    # Documented in monorepo/doc/pal/PalAdvancedProgrammingFunctions.md
    def rq_set_conveyor_clearance(is_left_pallet, height):
      if height < 0:
        popup("rq_set_conveyor_clearance(): The clearance height should be positive.", title="Palletizer", error=True,
        blocking=True)
      elif height == 0:
        height = 0.0001
      end

      pallet_side = "right"
      if(is_left_pallet):
         pallet_side = "left"
      end

      local palletId = node_rpc_server.getPalletId(pallet_side)
      node_rpc_server.setConveyorVerticalClearance(palletId, height)
    end
    ###############################################################
    # Linear Axis Move related methods
    ###############################################################
    def verify_is_in_linear_axis_range(target_axis_position):
      axis_position_range = node_rpc_server.linearaxisgetpositionrange()

      if target_axis_position < axis_position_range[0] or target_axis_position > axis_position_range[1]:
        textmsg("Linear axis target position : ", target_axis_position)
        textmsg("Linear axis position range : ", axis_position_range)
        popup("Linear axis position is unreachable.", "Linear Axis Move", blocking=True, error=True)
        halt
      end
    end

    # Documented in monorepo/doc/pal/PalAdvancedProgrammingFunctions.md
    def rq_get_linear_axis_pos():
        axis_position = node_rpc_server.linearaxisgetactualposition()
        return axis_position
    end

  BLOW_OFF_MODE_NO_AIR = 0
  BLOW_OFF_MODE_SMART_AIR = 1
  UNDEFINED_THREAD_ID = -1
  MODBUS_TYPE = "MODBUS"
  STANDARD_TYPE = "STANDARD"
  INVALID_OUTPUT_ADDRESS = -1
  RQ_UNUSED_TIMEOUT = -1

  global rq_cnc_insertion_node_ids = [-1, -1]
  global rq_run_timeout = 30

  ###################################################################################
  #
  # Generic methods
  #
  ###################################################################################

  def bool_to_str(value):
    if value:
      return "true"
    else:
      return "false"
    end
  end

  def bool_array_to_string(array, index):
    if (index >= length(array)):
      return "]"
    end

    separator = ","
    if (index == length(array) - 1):
      separator = ""
    end

    if (index == 0):
      str_array = concat("[", bool_to_str(array[index]), separator)
      return str_cat(str_array, bool_array_to_string(array, index + 1))
    else:
      return concat(bool_to_str(array[index]), separator, bool_array_to_string(array, index + 1))
    end
  end

  def rq_bool_array_to_string(array):
    return bool_array_to_string(array, 0)
  end

  def json_force_node(force, max_negative_deviation, max_positive_deviation, stiffness, enabled_axis, feature, is_adaptive):
    json = "{"
    json = concat(json, key_val("forceFrame", feature), ",")
    json = concat(json, key_val("isAdaptive", is_adaptive), ",")
    json = concat(json, key_val("isForceControlAboutActualPosition", "false"), ",")
    json = concat(json, key_val("isForceMode", enabled_axis), ",")
    json = concat(json, key_val("maxNegativeDeviation", max_negative_deviation), ",")
    json = concat(json, key_val("maxPositiveDeviation", max_positive_deviation), ",")
    json = concat(json, key_val("stiffness", stiffness), ",")
    json = concat(json, key_val("targetTcpWrench", force), "}")
    return json
  end

  def rq_setup_machine_tending_force_node(feature, force, stiffness, max_negative_deviation, max_positive_deviation, enabled_axis, is_adaptive):
    force_node_id = node_rpc_server.createnewforcenode()
    node_rpc_server.fromjson(force_node_id, json_force_node(force, max_negative_deviation, max_positive_deviation,
    stiffness, rq_bool_array_to_string(enabled_axis), 1, bool_to_str(is_adaptive)))
    return force_node_id
  end

  ###################################################################################
  #
  # TRAJECTORY UTILITIES
  #
  ###################################################################################

  def dot_product(v1, v2):
    return [v1]*transpose(v2)
  end

  def get_symmetric_poses_from_middle(p1, p2, middle_pose, distance):
    distance_p1_middle = point_dist(p1, middle_pose)
    alpha = (distance / 2) / distance_p1_middle
    start_pose = interpolate_pose(middle_pose, p1, alpha)
    end_pose = interpolate_pose(middle_pose, p2, alpha)

    return [start_pose, end_pose]
  end

  def translate_to_origin(pose):
    return p[0, 0, 0, pose[3], pose[4], pose[5]]
  end


  ###################################################################################
  #
  # ROBOTIQ PART PRESENTER
  #
  ###################################################################################

  global cnc_part_presenter_index = 0

  def rq_pallet_get_poses_from_index(p_corner_1_approach, p_corners, nb_rows, nb_columns, alternate_direction, index):
      row = floor(index / nb_columns)
      column = index % nb_columns

      row_alpha = 0
      if(nb_rows > 1):
          row_alpha = row / (nb_rows - 1)
      end

      p_row_start = interpolate_pose(p_corners[0], p_corners[3], row_alpha)
      p_row_end = interpolate_pose(p_corners[1], p_corners[2], row_alpha)

      column_alpha = 0
      if(nb_columns > 1):
          column_alpha = column / (nb_columns - 1)
      end

      if(alternate_direction and (row % 2) and nb_columns > 1):
          pallet_pose = interpolate_pose(p_row_end, p_row_start, column_alpha)
      else:
          pallet_pose = interpolate_pose(p_row_start, p_row_end, column_alpha)
      end

      T_1approach_1 = pose_trans(inv(p_corner_1_approach), p_corners[0])
      approach_pose = pose_trans(pallet_pose, inv(T_1approach_1))

      return [approach_pose, pallet_pose]
  end

  ###################################################################################
  #
  # MOVE DOOR
  #
  ###################################################################################

  def rq_setup_door_force_node(reference_frame, force, stiffness):
    feature = 1
    forces = [force,0,0,0,0,0]
    max_negative_deviation = [-5, 0, 0, 0, 0, 0]
    max_positive_deviation = [0.01, 0, 0, 0, 0, 0] # using a large value here would allow the trajectory to violate the kinematics limits, using zero removes the force node effect
    stiffnesses = [stiffness, 100, 100, 100, 100, 100]
    enabled_axis = [True, False, False, False, False, False]
    is_adaptive = True

    force_node_id = rq_setup_machine_tending_force_node(feature, forces, stiffnesses, max_negative_deviation,
    max_positive_deviation, enabled_axis, is_adaptive)

    node_rpc_server.setCustomFixedForceFrame(force_node_id, [reference_frame[3],reference_frame[4],reference_frame[5]])

    return force_node_id
  end

  def json_rq_moves_node(tcp_speed, tcp_accel):
    json = "{"
    json = concat(json, key_val("offsetType", 0), ",")
    json = concat(json, key_val("tcpSpeed", tcp_speed), ",")
    json = concat(json, key_val("tcpAccel", tcp_accel), ",")
    json = concat(json, key_val("actualreferenceframe", [0, 0, 0, 0, 0, 0]), ",")
    json = concat(json, key_val("originalreferenceframe", [0, 0, 0, 0, 0, 0]), "}")
    return json
  end

  def rq_setup_rqmoves_node(parent_node_id, tcp_speed, tcp_accel):
    rq_moves_node_id = node_rpc_server.createnewrqmoves()
    node_rpc_server.fromjson(rq_moves_node_id, json_rq_moves_node(tcp_speed, tcp_accel))
    node_rpc_server.setparentid(rq_moves_node_id, parent_node_id)
    return rq_moves_node_id
  end

  def rq_setup_waypoint_node(pose, joints, is_straight, parent_node_id):
    def json_waypoint_node(pose, joints, is_straight):
      json = "{"
      json = concat(json, key_val("jointPositions", joints), ",")
      json = concat(json, key_val("tcpPose", [pose[0],pose[1],pose[2],pose[3],pose[4],pose[5]]), ",")
      json = concat(json, key_val("isStraight", bool_to_str(is_straight)), "}")
      return json
    end

    waypoint_node_id = node_rpc_server.createnewwaypointnode()
    node_rpc_server.fromjson(waypoint_node_id, json_waypoint_node(pose, joints, is_straight))
    node_rpc_server.setparentid(waypoint_node_id, parent_node_id)
    node_rpc_server.rqmovesaddwaypoint(parent_node_id, waypoint_node_id)
    return waypoint_node_id
  end

  def rq_setup_move_door(reference_frame, start_pose, start_joints, stop_pose, stop_joints, move_force, contact_force, tcp_speed=0.4, tcp_accel=0.4):

    stop_pose_in_start_frame = pose_trans(pose_inv(start_pose), stop_pose)

    seeks_contact = False
    stiffness = 10
    move_force_node_id = rq_setup_door_force_node(reference_frame, move_force, stiffness)
    rq_moves_node_id = rq_setup_rqmoves_node(move_force_node_id, tcp_speed, tcp_accel)
    waypoint_open = rq_setup_waypoint_node(start_pose, start_joints, False, rq_moves_node_id)
    waypoint_close = rq_setup_waypoint_node(stop_pose, stop_joints, True, rq_moves_node_id)
    seeks_contact = True
    stiffness = 100
    contact_force_node_id = rq_setup_door_force_node(reference_frame, contact_force, stiffness)

    rq_movej_node_id = node_rpc_server.createnewmovejnode()
    node_rpc_server.setparentid(rq_movej_node_id, move_force_node_id)

    return [move_force_node_id, rq_moves_node_id, waypoint_open, waypoint_close, contact_force_node_id, rq_movej_node_id]
  end

  def rq_move_door(start_pose, start_joints, stop_pose, stop_joints, move_force, contact_force, tcp_speed, tcp_accel, approach_pose, approach_joints, end_reached_threshold=0.001):

    reference_frame = list_to_pose(kinematics_rpc_server.reorientP1WithXTowardP2andZApproxP1Z(start_pose, stop_pose))

    node_ids = rq_setup_move_door(reference_frame, start_pose, start_joints, stop_pose, stop_joints, move_force, contact_force, tcp_speed, tcp_accel)

    move_force_node_id = node_ids[0]
    rq_moves_node_id = node_ids[1]
    start_waypoint_node_id = node_ids[2]
    end_waypoint_node_id = node_ids[3]
    contact_force_node_id = node_ids[4]
    rq_movej_node_id = node_ids[5]

    rq_wait_ft_sensor_steady(2000)
    zero_ftsensor()
    sleep(0.1)

    path_answer = node_rpc_server.rqmovesinit(rq_moves_node_id)
    verify_path_answer(path_answer)

    approach_position_joints = get_inverse_kin(approach_pose, qnear=approach_joints)
    movej(approach_position_joints)

    node_rpc_server.movejdefinewaypoint(rq_movej_node_id, get_actual_joint_positions(), 1.0, 1.0)
    node_rpc_server.setparentid(rq_movej_node_id, move_force_node_id)
    reset_node_executor()
    active_and_reset_node(move_force_node_id)
    node_execution_thread = execute_node(rq_movej_node_id, True)

    path_answer = node_rpc_server.rqmovesinit(rq_moves_node_id)
    verify_path_answer(path_answer)
    q0 = node_rpc_server.rqmovesgetfirstpoint(rq_moves_node_id)
    node_rpc_server.setparentid(rq_movej_node_id, move_force_node_id)
    node_rpc_server.movejdefinewaypoint(rq_movej_node_id, q0, 1.0, 0.4)
    execute_node(rq_movej_node_id)
    execute_node(start_waypoint_node_id)
    execute_node(end_waypoint_node_id)

    kill_thread(node_execution_thread)

    node_rpc_server.movejdefinewaypoint(rq_movej_node_id, get_actual_joint_positions(), 1.0, 1.0)
    node_rpc_server.setparentid(rq_movej_node_id, contact_force_node_id)
    reset_node_executor()
    active_and_reset_node(contact_force_node_id)
    node_execution_thread = execute_node(rq_movej_node_id, True)

    timeout = 20
    while (point_dist(get_actual_tcp_pose(), stop_pose) > end_reached_threshold):
      if (timeout <= 0):
        popup("Door has not reached its final position")
        halt
      else:
        sync()
        timeout = timeout - get_steptime()
      end
    end

    kill_thread(node_execution_thread)

    approach_pose_in_start_frame = pose_trans(pose_inv(start_pose), approach_pose)
    retract_pose = pose_trans(get_actual_tcp_pose(), approach_pose_in_start_frame)
    movej(retract_pose)

    node_rpc_server.deletenode(move_force_node_id)
    node_rpc_server.deletenode(rq_moves_node_id)
    node_rpc_server.deletenode(start_waypoint_node_id)
    node_rpc_server.deletenode(end_waypoint_node_id)
    node_rpc_server.deletenode(contact_force_node_id)
    node_rpc_server.deletenode(rq_movej_node_id)

  end

  ###################################################################################
  #
  # CNC Insertion
  #
  ###################################################################################

  def rq_collet_insertion(contact_pose, insert_pose, inserted_pose):
      movel(contact_pose, a=1.2, v=0.025)
      movel(insert_pose, a=1.2, v=0.025)

      zero_ftsensor()
      sleep(0.1)

      direction = "Z+"
      stop_force_threshold = 3.0
      max_radius = 5.0
      radius_incr = 0.7
      peck_mode = False
      tangential_speed = 0.02
      compliant_insert_force_threshold = 10.0
      spiral_initial_pose_offset_name = "spiral_initial_pose_offset_name"
      rq_ins_destination = inserted_pose
      max_distance = point_dist(inserted_pose, get_actual_tcp_pose())
      rq_spiral_not_completed = False
      rq_ins_speed_setting = 0.02

      rq_insert_spiral_urcap(direction, stop_force_threshold, max_radius, radius_incr, peck_mode, tangential_speed, compliant_insert_force_threshold, spiral_initial_pose_offset_name)

      if (rq_spiral_not_completed):
        return False
      end

      return True
  end

  def rq_push_part(approach_pose, chuck_pose):
      zero_ftsensor()
      sleep(0.1)

      # Find pose with z axis pointing in the direction of the insertion
      p1 = translate_to_origin(approach_pose)
      insertion_dir_in_base_frame = pose_trans(p1, pose_trans(pose_inv(approach_pose), chuck_pose))
      ref_frame_pose = list_to_pose(kinematics_rpc_server.poseFromZaxis([insertion_dir_in_base_frame[0], insertion_dir_in_base_frame[1], insertion_dir_in_base_frame[2]]))

      surface_found = rq_linear_search_custom_frame("Z+", 10.0, 0.025, 0.1, ref_frame_pose)

      if not(surface_found):
          return False
      end

      return True
  end

  def rq_place_in_chuck(close_chuck_do, open_chuck_do, chuck_approach, chuck_position, chuck_delay):
      rq_open_workholding(close_chuck_do, open_chuck_do)

      movel(chuck_approach, a=1.2, v=0.25)
      movel(chuck_position, a=1.2, v=0.25)

      rq_close_workholding(close_chuck_do, open_chuck_do)
      sleep(chuck_delay)
  end

  def rq_pre_pick_in_chuck(chuck_approach, chuck_position, speed=0.25, accel=1.2):
      movel(chuck_approach, accel, speed)
      movel(chuck_position, accel, speed)
  end

  def rq_post_pick_in_chuck(close_chuck_do, open_chuck_do, chuck_approach, chuck_position, chuck_delay, speed=0.25,
  accel=1.2):
      rq_open_workholding(close_chuck_do, open_chuck_do)
      sleep(chuck_delay)

      movel(chuck_approach, accel, speed)
  end

  def rq_open_workholding(close_do, open_do):
      rq_set_workholding_do(close_do, open_do, False)
  end

  def rq_close_workholding(close_do, open_do):
      rq_set_workholding_do(close_do, open_do, True)
  end

  def rq_set_workholding_do(close_do, open_do, close_request):
      is_close_do_valid = rq_is_do_valid(close_do)
      is_open_do_valid = rq_is_do_valid(open_do)

      if(is_close_do_valid):
          set_standard_digital_out(close_do, close_request)
      end
      if(is_open_do_valid):
          set_standard_digital_out(open_do, not close_request)
      end
      if(is_close_do_valid or is_open_do_valid):
          sleep(0.5)
      end
  end

  def rq_is_do_valid(do_id):
      return do_id >= 0 and do_id <= 7
  end

  def set_cleaning_digital_output(address, state, blow_off_mode, output_type):
     if(blow_off_mode == BLOW_OFF_MODE_SMART_AIR):
       rq_set_output(output_type, address, state)
     end
  end

  ###################################################################################
  #
  # PATH GENERATOR 6 POINTS CURVE BUILT WITH 2 POINTS
  #
  ###################################################################################

  def execute_half_pipe(pose_1, pose_2,pose_transformation_air_nozzle_to_actual_tcp, depth, length_distance, width, angle, speed, spacing, address, output_type, blow_off_mode, passes):
    path_gen_poses = get_path_generator_6_points_poses(pose_1, pose_2, pose_transformation_air_nozzle_to_actual_tcp, depth, length_distance, width, angle)
    start_pose = p[path_gen_poses[0,0],path_gen_poses[0,1],path_gen_poses[0,2],path_gen_poses[0,3],path_gen_poses[0,4],path_gen_poses[0,5]]
    path_generator_node_id = setup_path_generator_6_points(path_gen_poses, speed, spacing)
    execute_path_generator_6_points(path_generator_node_id, start_pose,  address, output_type, blow_off_mode, passes)
  end

  def get_path_generator_6_points_poses(pose_2, pose_5,pose_transformation_air_nozzle_to_actual_tcp, depth=0.01, length=0, width=0.05, angle_deg=0):

    def offset_pose(pose, offset, offset_reference_frame, pose_transformation_air_nozzle_to_actual_tcp):
      pose_relative_to_ref_frame = express_pose_A_relative_to_pose_B(pose, offset_reference_frame)
      ref_frame_with_offset = pose_trans(offset_reference_frame, offset)
      pose_with_offset = pose_trans(ref_frame_with_offset, pose_relative_to_ref_frame)
      pose_with_offset_for_actual_tcp = pose_trans(pose_with_offset, pose_transformation_air_nozzle_to_actual_tcp)
      return pose_to_list(pose_with_offset_for_actual_tcp)
    end

    if(length > 0):
      middle_pose = interpolate_pose(pose_2, pose_5, 0.5)

      poses = get_symmetric_poses_from_middle(pose_2, pose_5, middle_pose, length)
      pose_2 = poses[0]
      pose_5 = poses[1]
    end

    path_ref_frame = list_to_pose(kinematics_rpc_server.reorientP1WithXTowardP2andZApproxP1Z(pose_2, pose_5))

    offset1 = pose_add(p[0,0,0,0,d2r(angle_deg),0], p[0, width,-depth,-d2r(angle_deg),0,0])
    offset2 = pose_add(p[0,0,0,0,d2r(angle_deg),0], p[0,     0,     0,              0,0,0])
    offset3 = pose_add(p[0,0,0,0,d2r(angle_deg),0], p[0,-width,-depth, d2r(angle_deg),0,0])

    pose_1_array = offset_pose(pose_2, offset1, path_ref_frame, pose_transformation_air_nozzle_to_actual_tcp)
    pose_2_array = offset_pose(pose_2, offset2, path_ref_frame, pose_transformation_air_nozzle_to_actual_tcp)
    pose_3_array = offset_pose(pose_2, offset3, path_ref_frame, pose_transformation_air_nozzle_to_actual_tcp)

    pose_4_array = offset_pose(pose_5, offset1, path_ref_frame, pose_transformation_air_nozzle_to_actual_tcp)
    pose_5_array = offset_pose(pose_5, offset2, path_ref_frame, pose_transformation_air_nozzle_to_actual_tcp)
    pose_6_array = offset_pose(pose_5, offset3, path_ref_frame, pose_transformation_air_nozzle_to_actual_tcp)

    return [pose_1_array, pose_2_array, pose_3_array, pose_4_array, pose_5_array, pose_6_array]
  end

  def setup_path_generator_6_points(pose_list, tcp_speed=0.1, spacing=0.02):

    def json_path_generator_node(pose_list, tcp_speed, spacing):

      SIX_POINTS_CURVE = 3
      OFFSET_TYPE_NONE = 0
      FORCE_OPPOSITE_SIDE = 2

      json = "{"
      json = concat(json, key_val("tcpSpeed", tcp_speed), ",")
      json = concat(json, key_val("poses", pose_list), ",")
      json = concat(json, key_val("avoidAbruptEnd", "false"), ",")
      json = concat(json, key_val("isSurfaceFillOn", "true"), ",")
      json = concat(json, key_val("spacing", spacing), ",")
      json = concat(json, key_val("pathType", SIX_POINTS_CURVE), ",")
      json = concat(json, key_val("offsetType",OFFSET_TYPE_NONE), ",")
      json = concat(json, key_val("endingMode", FORCE_OPPOSITE_SIDE), "}")

      return json
    end

    rq_path_generator_parent_id = 0
    path_generator_node_id = node_rpc_server.createPathGeneratorNode()
    node_rpc_server.fromjson(path_generator_node_id, json_path_generator_node(pose_list, tcp_speed, spacing))
    node_rpc_server.setparentid(path_generator_node_id, rq_path_generator_parent_id)

    return path_generator_node_id
  end

  def execute_path_generator_6_points(path_generator_node_id, pose_1, address = INVALID_OUTPUT_ADDRESS, output_type = MODBUS_TYPE, blow_off_mode = BLOW_OFF_MODE_NO_AIR, passes = 1):
    index = 0
    while (index < passes):
      movej(get_inverse_kin(pose_1))
      set_cleaning_digital_output(address, True, blow_off_mode, output_type)
      reset_node_executor()
      node_execution_thread = execute_node(path_generator_node_id, True)
      rq_continue_node_execution = False
      set_cleaning_digital_output(address, False, blow_off_mode, output_type)
      join node_execution_thread
      index = index + 1
    end
    node_rpc_server.deletenode(path_generator_node_id)
  end

  ###################################################################################
  #
  # Straight line trajectory
  #
  ###################################################################################

  def execute_straight_line(p1, p2,pose_transformation_air_nozzle_to_actual_tcp, accel=1.2, speed=0.25, distance = 0, angles = [0, 0, 0], address = INVALID_OUTPUT_ADDRESS, output_type = MODBUS_TYPE, blow_off_mode = BLOW_OFF_MODE_NO_AIR, passes = 1):
    offset_for_angles = p[0, 0, 0, d2r(angles[0]), d2r(angles[1]), d2r(angles[2])]
    p1 = pose_trans(p1, offset_for_angles)
    p2 = pose_trans(p2, offset_for_angles)

    # apply transformation to take into account that the actual tcp offset is not the same as the one that was used when the waypoints were saved:
    p1 = pose_trans(p1, pose_transformation_air_nozzle_to_actual_tcp)
    p2 = pose_trans(p2, pose_transformation_air_nozzle_to_actual_tcp)
    global air_output_adress = address

    qActual = get_actual_joint_positions()
    CleanPathId = node_rpc_server.createnewcleaningpathnode(p1, p2, qActual, passes, distance, accel, speed, blow_off_mode)

    reset_node_executor()
    if output_type == MODBUS_TYPE:
      air_thread = run modbusAirControlThread()
    elif output_type == STANDARD_TYPE:
      air_thread = run standardAirControlThread()
    end

    node_execution_thread = execute_node(CleanPathId, True)
    rq_continue_node_execution = False

    join node_execution_thread
    node_rpc_server.deletenode(CleanPathId)
    if output_type == MODBUS_TYPE or output_type == STANDARD_TYPE :
      kill air_thread
    end
  end

  ###################################################################################
  #
  # Cross trajectory
  #
  ###################################################################################

  def find_cross_trajectory_poses(p1, p2, height=0, width=0, p1_angles = [0, 0, 0], p2_angles = [0, 0, 0], p3_angles = [0, 0, 0], p4_angles = [0, 0, 0]):
    def find_side_poses(p0, p1):
      def find_side_pose(p0,p1,angle):
        p1_T_p0 = pose_trans(pose_inv(p0), p1)
        rotated_p0_by_90_degrees = pose_trans(p0, p[0, 0, 0, 0, 0, d2r(angle)])

        side_pose = pose_trans(rotated_p0_by_90_degrees, p1_T_p0)
        side_pose[3] = p0[3]
        side_pose[4] = p0[4]
        side_pose[5] = p0[5]

        return side_pose
      end

      p3= find_side_pose(p0, p1, 90)
      p4 = find_side_pose(p0, p1, 270)

      return [p3, p4]
    end

    def get_start_and_end_poses_based_on_distance(p1, p2, middle_pose, distance):
      if(distance == 0):
        start_pose = p1
        end_pose = p2
      else:
        poses = get_symmetric_poses_from_middle(p1, p2, middle_pose, distance)
        start_pose = poses[0]
        end_pose = poses[1]
      end
      return [start_pose, end_pose]
    end

    def get_side_poses_based_on_distance(p1, p2, middle_pose, width):
      if(width == 0):
        side_poses = find_side_poses(middle_pose, p1)
      else:
        poses = get_symmetric_poses_from_middle(p1, p2, middle_pose, width)
        side_poses = find_side_poses(middle_pose, poses[0])
      end

      return side_poses
    end

    def get_angle_offset(angles):
      return  p[0, 0, 0, d2r(angles[0]), d2r(angles[1]), d2r(angles[2])]
    end

    middle_pose = interpolate_pose(p1, p2, 0.5)

    start_and_end_poses = get_start_and_end_poses_based_on_distance(p1, p2, middle_pose, height)
    side_poses = get_side_poses_based_on_distance(p1, p2, middle_pose, width)

    p1_offset = get_angle_offset(p1_angles)
    p2_offset = get_angle_offset(p2_angles)
    p3_offset = get_angle_offset(p3_angles)
    p4_offset = get_angle_offset(p4_angles)

    start_and_end_poses[0] = pose_trans(start_and_end_poses[0], p1_offset)
    start_and_end_poses[1] = pose_trans(start_and_end_poses[1], p2_offset)
    side_poses[0] = pose_trans(side_poses[0], p3_offset)
    side_poses[1] = pose_trans(side_poses[1], p4_offset)

    return [middle_pose, start_and_end_poses[0], start_and_end_poses[1], side_poses[0], side_poses[1]]
  end

  def execute_cross_trajectory(p1, p2,pose_transformation_air_nozzle_to_actual_tcp, height=0, width=0, p1_angles = [0, 0, 0], p2_angles = [0, 0, 0], p3_angles = [0, 0, 0], p4_angles = [0, 0, 0], accel=1.2, speed=0.25,  address = INVALID_OUTPUT_ADDRESS, output_type = MODBUS_TYPE, blow_off_mode = BLOW_OFF_MODE_NO_AIR, passes = 1):

    cross_poses = find_cross_trajectory_poses(p1, p2, height, width, p1_angles, p2_angles, p3_angles, p4_angles)

    p0 = pose_trans(cross_poses[0], pose_transformation_air_nozzle_to_actual_tcp)
    p1 = pose_trans(cross_poses[1], pose_transformation_air_nozzle_to_actual_tcp)
    p2 = pose_trans(cross_poses[2], pose_transformation_air_nozzle_to_actual_tcp)
    p3 = pose_trans(cross_poses[3], pose_transformation_air_nozzle_to_actual_tcp)
    p4 = pose_trans(cross_poses[4], pose_transformation_air_nozzle_to_actual_tcp)

   index = 0

   while (index < passes):
     movej(get_inverse_kin(p0))
     set_cleaning_digital_output(address, True, blow_off_mode, output_type)
     movel(p1, accel, speed)
     movel(p2, accel, speed)
     movel(p0, accel, speed)
     movel(p3, accel, speed)
     movel(p4, accel, speed)
     set_cleaning_digital_output(address, False, blow_off_mode, output_type)
     index = index + 1
   end
  end

  def execute_waypoint_cross_trajectory(starting_pose, finishing_pose, accel=1.2, speed=0.25):
   movej(get_inverse_kin(starting_pose))
   movel(finishing_pose, accel, speed)
  end

  ###################################################################################
  #
  # Fermat spiral trajectory
  #
  ###################################################################################

  def execute_fermat_spiral(start_pose, end_pose,pose_transformation_air_nozzle_to_actual_tcp, max_radius = 0, angle = 0, number_of_turns = 1, speed = 0.25,address = INVALID_OUTPUT_ADDRESS, output_type = MODBUS_TYPE, blow_off_mode = BLOW_OFF_MODE_NO_AIR, passes = 1):
    def find_middle(start_pose, end_pose):
      alpha = 0.5
      return interpolate_pose(start_pose, end_pose, alpha)
    end

    def find_next_theta(spiral_constant, theta, speed):
      denom = spiral_constant * sqrt(1/(4*theta) + theta)
      theta_dot = speed / denom
      theta = theta + theta_dot * rq_controller_time_step
      return theta
    end

    def find_spiral_pose(theta, spiral_plane, center_pose, angle, spiral_constant, pose_transformation_air_nozzle_to_actual_tcp):
      local r = spiral_constant * sqrt(theta)
      local x = r * cos(theta)
      local y = r * sin(theta)

      local p2 = pose_trans(spiral_plane, p[x,y,0,0,0,0])
      local p3 = p[p2[0], p2[1], p2[2], center_pose[3], center_pose[4], center_pose[5]]
      local p4 = pose_trans(p3, pose_transformation_air_nozzle_to_actual_tcp)
      local p5 = pose_trans(p4, p[0, 0, 0, -d2r(angle)*cos(theta), -d2r(angle)*sin(theta), 0])
      return p5
    end

    def execute_outer_to_inner_spiral(start_pose, middle_pose, spiral_plane, pose_transformation_air_nozzle_to_actual_tcp, max_angle, angle, spiral_constant_nominal, speed, address, output_type, blow_off_mode):
      local theta = max_angle
      local max_r = point_dist(start_pose, middle_pose)
      local spiral_constant = -1 * spiral_constant_nominal
      local r = max_r
      local is_first_pose = True

      while (norm((r)) <= max_r):
        theta = find_next_theta(spiral_constant, theta, speed)
        if(theta < 0):
          break
        end

        r = spiral_constant * sqrt(theta)
        next_pose = find_spiral_pose(theta, spiral_plane, middle_pose, angle, spiral_constant, pose_transformation_air_nozzle_to_actual_tcp)

        if (is_first_pose):
          movej(get_inverse_kin(next_pose))
          set_cleaning_digital_output(address, True, blow_off_mode, output_type)
          is_first_pose = False
        else:
          servoj(get_inverse_kin(next_pose), t = rq_controller_time_step)
        end
      end
    end

    def execute_inner_to_outer_spiral(start_pose, middle_pose, spiral_plane, pose_transformation_air_nozzle_to_actual_tcp, angle, spiral_constant, speed):
      local theta = 0.0001
      local max_r = point_dist(start_pose, middle_pose)
      local r = 0

      while (norm(r) <= max_r):
        theta = find_next_theta(spiral_constant, theta, speed)
        r = spiral_constant * sqrt(theta)
        next_pose = find_spiral_pose(theta, spiral_plane, middle_pose, angle, spiral_constant, pose_transformation_air_nozzle_to_actual_tcp)
        servoj(get_inverse_kin(next_pose), t = rq_controller_time_step)
      end
    end

    max_angle = d2r(number_of_turns * 360)
    middle_pose = find_middle(start_pose, end_pose)

    if(max_radius > 0):
      poses = get_symmetric_poses_from_middle(start_pose, end_pose, middle_pose, max_radius * 2)
      start_pose = poses[0]
      end_pose = poses[1]
    end

    SPIRAL_CONSTANT = (point_dist(middle_pose, start_pose)) / sqrt(max_angle)

    spiral_plane = list_to_pose(kinematics_rpc_server.reorientP1WithXTowardP2andZApproxP1Z(middle_pose, end_pose))


    index = 0
    while(index < passes):
      execute_outer_to_inner_spiral(start_pose, middle_pose, spiral_plane,pose_transformation_air_nozzle_to_actual_tcp, max_angle, angle, SPIRAL_CONSTANT, speed, address, output_type, blow_off_mode)
      execute_inner_to_outer_spiral(end_pose, middle_pose, spiral_plane, pose_transformation_air_nozzle_to_actual_tcp, angle, SPIRAL_CONSTANT, speed)
      set_cleaning_digital_output(address, False, blow_off_mode, output_type)
      index = index + 1
    end
  end

  ###################################################################################
  #
  # ROBOTIQ VISE INSERTION
  #
  # - The first touch is performed in the direction of the gravity, regardless of
  #   the robot mounting orientation, tcp offset and TCP orientation
  # - Optional 2e et 3e touch are performed relative to TCP. They require that, at
  #   the moment that the insertion is performed, the TCP is oriented such that one
  #   axis is aligned with the gravity. The TCP axes for the 2e and 3e touch are
  #   chosen as the ones not aligned with the gravity.
  ###################################################################################
  def insert_in_vise(start_pose, end_pose, number_of_touch=3, forces=[10, 20, 20], invert_axis=False, move_to_end_pose=False):

    def list_by_scalar_multiply_(l1, scalar):
      result = l1
      i=0
      while i<length(result):
        result[i]=l1[i]*scalar
        i=i+1
      end
      return result
    end

    def find_gravity_direction(acceleration_direction, threshold):
      result = [False, False, False]
      i = 0
      while i < length(result):
        result[i] =  norm(acceleration_direction[i]) > threshold
        i = i + 1
      end
      return result
    end

    def get_axis(index, direction):
      axis = "XYZ"
      if direction < 0:
        sign = "-"
      elif direction > 0:
        sign = "+"
      else:
        popup("insert_in_vise:get_axis >>> direction cannot be 0. Fix it.")
        halt
      end
      return str_cat(str_sub(axis, index, 1), sign)
    end

    def direction_to_index(str):
      if "X" == str_sub(str, 0, 1):
        return 0
      elif "Y" == str_sub(str, 0, 1):
        return 1
      elif "Z" == str_sub(str, 0, 1):
        return 2
      else:
        popup("invalid direction :", str)
        halt
      end
    end

    def find_touch_direction(mask, direction):
      i = 0
      result = [0, 0, 0]
      while i < 3:
        if mask[i]:
          result[i] = direction[i]
        end
        i = i + 1
      end
      return result
    end

    def find_touch_direction_str(mask, direction):
      i = 0
      result = ""
      while i < 3:
        if mask[i]:
          result = str_cat(result, get_axis(i, direction[i]))
        end
        i = i + 1
      end
      return result
    end

    def invert(list):
      result = list
      i = 0
      while i < length(list):
        result[i] = not list[i]
        i = i + 1
      end
      return result
    end

    def assert_that_the_first_touch_is_aligned_with_an_axis(first_touch_direction_mask):
      i = 0
      counter = 0
      while i < length(first_touch_direction_mask):
        if first_touch_direction_mask[i]:
          counter = counter + 1
        end
        i = i + 1
      end

      if counter != 1:
        popup("One of the TCP axes must be perpendicular to the floor while loading the part in the vise.")
        halt
      end
    end

    def setup_nodes(forces, number_of_touch, first_touch_direction_mask, direction, second_direction_str, third_direction_str):
      def max_deviation_from(forces, enabled_axis):
        i = 0
        deviation = [0, 0, 0, 0, 0, 0]
        while i < 3:
          if forces[i] > 0:
            deviation[i] = 10
          elif forces[i] ==  0:
            deviation[i] = 10
          end
          i = i + 1
        end
        while i < 6:
          if enabled_axis[i]:
            deviation[i] = 0.35
          end
          i = i + 1
        end
        return deviation
      end

      def min_deviation_from(forces, enabled_axis):
        i = 0
        deviation = [0, 0, 0, 0, 0, 0]
        while i < 3:
          if forces[i] < 0:
            deviation[i] = -10
          elif forces[i] ==  0:
            deviation[i] = -10
          end
          i = i + 1
        end
        while i < 6:
          if enabled_axis[i]:
            deviation[i] = -0.35
          end
          i = i + 1
        end
        return deviation
      end

      def stiffness_from(forces):
        i = 0
        stiffness = [0, 0, 0, 100, 100, 100]
        while i < length(forces):
          if norm(forces[i]) > 0:
            stiffness[i] = 100
          else:
            stiffness[i] = 85
          end
          i = i + 1
        end
        return stiffness
      end

      def compute_final_forces(forces, number_of_touch, first_touch_direction_mask, direction, second_direction_str, third_direction_str):
        final_forces = [0, 0, 0]
        if number_of_touch > 0:
          i = 0
          while i < length(first_touch_direction_mask):
            if first_touch_direction_mask[i]:
              break
            end
            i = i + 1
          end
          final_forces[i] = direction[i] * forces[i]
        end
        if number_of_touch > 1:
          i = direction_to_index(second_direction_str)
          final_forces[i] = direction[i] * forces[i]
        end
        if number_of_touch > 2:
          i = direction_to_index(third_direction_str)
          final_forces[i] = direction[i] * forces[i]
        end
        return final_forces
      end

      def compute_enabled_axis(first_touch_direction_mask):
        enabled_axis = [True, True, True, False, False, False]
        i = 0
        while i < length(first_touch_direction_mask):
          if first_touch_direction_mask[i]:
            break
          end
          i = i + 1
        end
        enabled_axis[i + 3] = True

        return enabled_axis
      end

      final_forces = compute_final_forces(forces, number_of_touch, first_touch_direction_mask, direction, second_direction_str, third_direction_str)
      enabled_axis = compute_enabled_axis(first_touch_direction_mask)

      force_node_id = rq_setup_machine_tending_force_node(1, [final_forces[0], final_forces[1], final_forces[2], 0, 0, 0], stiffness_from
      (final_forces), min_deviation_from(final_forces, enabled_axis), max_deviation_from(final_forces, enabled_axis),
      enabled_axis, False)
      movej_node_id = node_rpc_server.createnewmovejnode()
      node_rpc_server.setparentid(movej_node_id, force_node_id)

      return [force_node_id, movej_node_id]
    end

    def average_tool_acceleration_reading(n_samples, delay):
      n = n_samples
      reading = [0, 0, 0]
      while n > 0:
        reading = reading + get_tool_accelerometer_reading()
        sleep(delay)
        n = n - 1
      end
      return reading/n_samples
    end

    def linear_search_toward_gravity(force):
      # maybe add a stopj here to prevent acceleration reading to be influenced by robot movement
      flange_accel = average_tool_acceleration_reading(10, 0.1) # measured accel is oriented in gravity oposite direction
      flange_accel_pose = p[-flange_accel[0], -flange_accel[1], -flange_accel[2], 0, 0,0]
      p1 = translate_to_origin(get_actual_tool_flange_pose())
      gravity_dir_in_base_frame = pose_trans(p1, flange_accel_pose)

      # Find pose with z axis pointing in gravity direction:
      ref_frame_pose = list_to_pose(kinematics_rpc_server.poseFromZaxis([gravity_dir_in_base_frame[0], gravity_dir_in_base_frame[1], gravity_dir_in_base_frame[2]]))
      speed = 0.01
      abs_max_distance = 0.05

      surface_found = rq_linear_search_custom_frame("Z+", force, speed, abs_max_distance, ref_frame_pose)
      return surface_found
    end

    #### Actual insert_in_vise method ####
    movel(start_pose)
    zero_ftsensor()

    # 1. Use accelerometer reading to find touches directions:
    ACCELERATION_THRESHOLD = 8
    flange_accel = average_tool_acceleration_reading(10, 0.1)
    tcp_accel = pose_trans(pose_inv(get_tcp_offset()), p[flange_accel[0], flange_accel[1], flange_accel[2], 0, 0, 0])
    first_touch_direction_mask = find_gravity_direction(tcp_accel, ACCELERATION_THRESHOLD)
    assert_that_the_first_touch_is_aligned_with_an_axis(first_touch_direction_mask)

    direction_transform = pose_trans(pose_inv(start_pose), end_pose)
    direction = [direction_transform[0], direction_transform[1], direction_transform[2]]
    direction_sign = [direction[0]/norm(direction[0]), direction[1]/norm(direction[1]), direction[2]/norm(direction[2])]

    touch_direction_str = find_touch_direction_str(invert(first_touch_direction_mask), direction_sign)
    touch_direction = find_touch_direction(invert(first_touch_direction_mask), direction_sign)

    if invert_axis:
      second_direction_str = str_sub(touch_direction_str, 0, 2)
      third_direction_str = str_sub(touch_direction_str, 2, 4)
    else:
      second_direction_str = str_sub(touch_direction_str, 2, 4)
      third_direction_str = str_sub(touch_direction_str, 0, 2)
    end

    end_pose_orientation = translate_to_origin(end_pose)

    # 2. Prepare nodes:
    rq_cnc_insertion_node_ids = setup_nodes(forces, number_of_touch, first_touch_direction_mask, direction_sign, second_direction_str, third_direction_str)
    feature_tool = 1

    # 3. Perform touches:
    if number_of_touch > 0:
      surface_found = linear_search_toward_gravity(forces[0])
      if not surface_found:
        textmsg("Insertion in vise: First contact has not been found")
        popup("First contact has not been found", title="Insertion in vise", blocking=True)
        return UNDEFINED_THREAD_ID
      end
    end
    if number_of_touch > 1:
      surface_found = rq_linear_search_urcap(second_direction_str, forces[1], 0.01, 0.05, feature_tool)
      if not surface_found:
        textmsg("Insertion in vise: Second contact has not been found")
        popup("Second contact has not been found", title="Insertion in vise", blocking=True)
        return UNDEFINED_THREAD_ID
      end
    end
    if number_of_touch > 2:
      surface_found = rq_linear_search_urcap(third_direction_str, forces[2], 0.01, 0.05, feature_tool)
      if not surface_found:
        textmsg("Insertion in vise: Third contact has not been found")
        popup("Third contact has not been found", title="Insertion in vise", blocking=True)
        return UNDEFINED_THREAD_ID
      end
    end

    # 4. Move to end position:
    if not move_to_end_pose:
      end_pose = get_actual_tcp_pose()
    end

    node_rpc_server.movejdefinewaypoint(rq_cnc_insertion_node_ids[1], get_actual_joint_positions(), 1.0, 1.0)
    reset_node_executor()
    active_and_reset_node(rq_cnc_insertion_node_ids[0])
    node_execution_thread = execute_node(rq_cnc_insertion_node_ids[1], True)
    node_rpc_server.movejdefinewaypoint(rq_cnc_insertion_node_ids[1], get_inverse_kin(end_pose), 1.0, 1.0)
    execute_node(rq_cnc_insertion_node_ids[1])
    sleep(1)
    return node_execution_thread
  end

  ###################################################################################
  # AIR OUTPUT CONTROL
  ###################################################################################
  thread modbusAirControlThread():
    while (True):
      rq_air_value = read_input_boolean_register(101)
      modbus_set_output_signal(air_output_adress, rq_air_value, False)
      sleep(rq_controller_time_step)
    end
  end

  thread standardAirControlThread():
    while (True):
      rq_air_value = read_input_boolean_register(101)
      set_digital_out(air_output_adress, rq_air_value)
      sleep(rq_controller_time_step)
    end
  end
  def rq_set_output(output_type, address, value):
    if output_type == "MODBUS":
      modbus_set_output_signal(address, value)
    elif output_type == "STANDARD":
      set_standard_digital_out(address, value)
    end
  end

  def rq_digital_output_action(action, output_type, address, time_on=1, time_off=0.5, delay_after=0):
    if action == "PUSH_AND_HOLD":
      rq_set_output(output_type, address, True)
    elif action == "PUSH":
      rq_set_output(output_type, address, True)
      sleep(time_on)
      rq_set_output(output_type, address, False)
    elif action == "DOUBLE_PUSH":
      rq_set_output(output_type, address, True)
      sleep(time_on)
      rq_set_output(output_type, address, False)
      sleep(time_off)
      rq_set_output(output_type, address, True)
      sleep(time_on)
      rq_set_output(output_type, address, False)
    elif action == "RELEASE":
      rq_set_output(output_type, address, False)
    end
    sleep(delay_after)
  end
  def json_kinematic_parameters_ratio(ratio):
    json = "{"
    json = concat(json, key_val("kinematicParametersRatio", ratio), "}")
    return json
  end

  def execute_move_along_trail(trail_node_id, joint_positions, kinematic_parameters_ratio):
    node_rpc_server.fromjson(trail_node_id, json_kinematic_parameters_ratio(kinematic_parameters_ratio))
    roadmap_state = node_rpc_server.initRoadmap(trail_node_id, joint_positions)
    path_time = roadmap_state[0]

    if(path_time > 0.0):
      reset_node_executor()
      node_execution_thread = execute_node(trail_node_id, True)
      kill node_execution_thread
    end
  end
    global servojId = 2
  rq_collision_detection_stop()
  # end: URCap Installation Node
  global timer_1=0
  global c1_p=p[.157577147953, -.388190086959, .151522802335, -3.141047500236, -.055722937685, .000049173003]
  global c1_q=[-0.8664591948138636, -1.9946533642210902, -1.2442758083343506, -1.4727600377849122, 1.5722702741622925, 3.80899977684021]
  global Waypoint_8_p=p[-.150427162654, -.390225762120, .151546909862, -3.141036571135, -.055876152350, -.000047259053]
  global Waypoint_8_q=[-1.6194260756122034, -1.9913011989989222, -1.2490886449813843, -1.4713011544993897, 1.5722861289978027, 3.055936574935913]
  global Waypoint_9_p=p[-.150708861961, -.348227279771, .151556678779, -3.140981415271, -.055839736306, -.000005615584]
  global Waypoint_9_q=[-1.6259835402118128, -1.8204313717284144, -1.484473705291748, -1.4068395358375092, 1.5721334218978882, 3.049475908279419]
  global c2_p=p[.157334690756, -.346187468466, .151541407059, -3.140997979648, -.055849351266, -.000096657697]
  global c2_q=[-0.7918246428119105, -1.8239737949767054, -1.4800207614898682, -1.4076639872840424, 1.5722535848617554, 3.8836276531219482]
  global c3_p=p[.157083701424, -.312184047431, .151537015881, -3.141022089074, -.055797227736, -.000052619000]
  global c3_q=[-0.7196467558490198, -1.6905099354186, -1.6421176195144653, -1.379027785067894, 1.572106122970581, 3.9558956623077393]
  global Waypoint_11_p=p[-.150940969920, -.314230691157, .151536383906, -3.140942113866, -.055656910778, .000084669065]
  global Waypoint_11_q=[-1.6325328985797327, -1.686746736566061, -1.6463444232940674, -1.3786910337260743, 1.5719581842422485, 3.0430991649627686]
  global Waypoint_10_p=p[-.151215527839, -.272202295578, .151528000621, -3.140750457776, -.055565181978, -.000054283277]
  global Waypoint_10_q=[-1.642848316823141, -1.5211668771556397, -1.818166971206665, -1.37264800191436, 1.5718692541122437, 3.0329036712646484]
  global c4_p=p[.156798309975, -.270188328283, .151523853386, -3.140995537507, -.055867543787, -.000025290066]
  global c4_q=[-0.6114972273456019, -1.5255678755095978, -1.8141570091247559, -1.371950702076294, 1.5719618797302246, 4.064064025878906]
  global chipC_p=p[-.099700577098, -.183627440197, .208433402457, 3.139691259007, -.105394058226, -.000149781669]
  global chipC_q=[-1.3891781012164515, -1.0096948903850098, -1.88504958152771, -1.8167749843993128, 1.5708818435668945, 3.388993501663208]
  global Waypoint_15_p=p[-.099704296715, -.202951379992, .208432580258, 3.139670120847, -.105426183766, -.000160358536]
  global Waypoint_15_q=[-1.4082286993609827, -1.099871740942337, -1.8470300436019897, -1.764597078362936, 1.5709946155548096, 3.369927167892456]
  global Waypoint_25_p=p[-.122879871442, -.368965239733, .188211838452, 3.139821275232, -.105433326911, -.000075080205]
  global Waypoint_25_q=[-1.5479124228106897, -1.8512498341002406, -1.271846055984497, -1.5885349712767542, 1.5719534158706665, 3.2300467491149902]
  global Waypoint_26_p=p[-.293995928019, -.360529248638, .222497263242, 3.139820833490, -.105446172100, -.000068418500]
  global Waypoint_26_q=[-1.9689658323871058, -2.3604399166502894, -0.28896433115005493, -2.062209268609518, 1.571913719177246, 2.8087823390960693]
  global Waypoint_27_p=p[-.293996037589, -.360524548960, .073401623062, -3.139818121402, .105463968189, .000065100461]
  global Waypoint_27_q=[-1.9687660376178187, -2.2716170750060023, -1.1700339317321777, -1.2699676317027588, 1.5726664066314697, 2.809603691101074]
  global Waypoint_28_p=p[-.293994929318, -.360517570897, .073396573982, -3.079220194370, .622813891331, .000072005146]
  global Waypoint_28_q=[-1.9687660376177893, -2.2716089687261967, -1.1700649262597302, -1.269964114900139, 1.572658061981124, 3.141592653589793]
  global Waypoint_29_p=p[-.293994178547, -.360515134427, .073402631236, -3.140584062493, .078656845609, .000054923880]
  global Waypoint_29_q=[-1.9687698523153152, -2.2715932331392654, -1.1700625419823325, -1.2699834567121284, 1.5726652145390896, 2.792526803190927]
  global Waypoint_30_p=p[-.293991359760, -.360511345669, .073405660262, -3.079212155022, .622831433047, .000021425167]
  global Waypoint_30_q=[-1.9687779585452905, -2.271581312216341, -1.170064806944243, -1.2700025898209706, 1.5726886987653534, 3.141592653589793]
  global Waypoint_31_p=p[-.293995928019, -.360529248638, .222497263242, 3.139820833490, -.105446172100, -.000068418500]
  global Waypoint_31_q=[-1.9689658323871058, -2.3604399166502894, -0.28896433115005493, -2.062209268609518, 1.571913719177246, 2.8087823390960693]
  global Waypoint_32_p=p[-.120064390322, -.465070651334, .187365924664, 2.700279766902, -.088400420341, .019763045538]
  global Waypoint_32_q=[-1.5412524382220667, -1.9475652180113734, -1.406833291053772, -0.9173591893962403, 1.5603561401367188, 3.2332537174224854]
  global Waypoint_33_p=p[-.125099110421, -.299097154487, .189878767902, 3.139750209928, -.105401717856, -.000111797080]
  global Waypoint_33_q=[-1.550074879323141, -1.5617311683348198, -1.5979981422424316, -1.5518303674510499, 1.5716702938079834, 3.2279696464538574]
  global Waypoint_1_p=p[.263501689877, -.337317763427, .239349489480, 3.139797243720, -.105347053477, -.000037720516]
  global Waypoint_1_q=[-0.5959728399859827, -2.1057659588255824, -0.6533136367797852, -1.9525557957091273, 1.5718059539794922, 4.181682586669922]
  global Waypoint_2_p=p[.265438435610, -.352444474661, .141740907029, 3.139726376264, -.105360108121, -.000022031768]
  global Waypoint_2_q=[-0.6231134573565882, -2.1016999683775843, -1.126999020576477, -1.4828875821879883, 1.5722739696502686, 4.154912948608398]
  global Waypoint_3_p=p[.206441973084, -.349241721273, .141737893294, 3.139734184252, -.105329347268, -.000022485776]
  global Waypoint_3_q=[-0.7073677221881312, -1.9410401783385218, -1.3681066036224365, -1.4024366003325959, 1.5721865892410278, 4.070710182189941]
  global Waypoint_4_p=p[.157616611756, -.378012026932, .141738203587, 3.139764187573, -.105376653239, -.000076760662]
  global Waypoint_4_q=[-0.8494070211993616, -1.9579774341978968, -1.3439116477966309, -1.409730003481247, 1.5722019672393799, 3.928692579269409]
  global Waypoint_5_p=p[.109134761588, -.393436595889, .141742225598, 3.139732501163, -.105376381431, -.000050533951]
  global Waypoint_5_q=[-0.972816292439596, -1.9523960552611292, -1.3519116640090942, -1.4072665137103577, 1.5721949338912964, 3.805286407470703]
  global Waypoint_6_p=p[-.188131250090, -.345166366147, .141750553976, 3.139727051239, -.105353578209, -.000024875816]
  global Waypoint_6_q=[-1.7293437162982386, -1.8864180050291957, -1.4439769983291626, -1.381135032778122, 1.572224736213684, 3.0487747192382812]
  global Waypoint_7_p=p[-.131564048097, -.216205376465, .141741700579, 3.139714533984, -.105382776464, -.000044168049]
  global Waypoint_7_q=[-1.572542969380514, -1.2417927545360108, -2.0833356380462646, -1.3863917154124756, 1.571577787399292, 3.2058310508728027]
  global timer_1_is_counting=False
  thread Timer_Thread():
    while (True):
      if (timer_1_is_counting):
        timer_1 = timer_1 + get_steptime()
      end
      sync()
    end
  end
  run Timer_Thread()
  def Spraychip2():
    $ 372 "Spraychip2" "noBreak"
    $ 373 "MoveJ"
    $ 374 "chipC" "breakAfter"
    movej(get_inverse_kin(chipC_p, qnear=chipC_q), a=1.3962634015954636, v=1.0471975511965976)
    $ 375 "c≔chipC"
    global c=chipC_p
    $ 376 "rc≔27/1000"
    global rc=27/1000
    $ 377 "p0≔p[c[0]+rc,c[1],c[2],c[3],c[4],c[5]-1.5*0]"
    global p0=p[c[0]+rc,c[1],c[2],c[3],c[4],c[5]-1.5*0]
    $ 378 "p45≔p[c[0]+0.71*rc,c[1]+0.71*rc,c[2],c[3]-0/1.1,c[4],c[5]-0/1.1]"
    global p45=p[c[0]+0.71*rc,c[1]+0.71*rc,c[2],c[3]-0/1.1,c[4],c[5]-0/1.1]
    $ 379 "p90≔p[c[0],c[1]+rc,c[2],c[3]-0,c[4],c[5]]"
    global p90=p[c[0],c[1]+rc,c[2],c[3]-0,c[4],c[5]]
    $ 380 "p135≔p[c[0]-0.71*rc,c[1]+0.71*rc,c[2],c[3]-0/1.1,c[4],c[5]+0/1.1]"
    global p135=p[c[0]-0.71*rc,c[1]+0.71*rc,c[2],c[3]-0/1.1,c[4],c[5]+0/1.1]
    $ 381 "p180≔p[c[0]-rc,c[1],c[2],c[3],c[4],c[5]+1.5*0]"
    global p180=p[c[0]-rc,c[1],c[2],c[3],c[4],c[5]+1.5*0]
    $ 382 "p225≔p[c[0]-0.71*rc,c[1]-0.71*rc,c[2],c[3]+0/1.1,c[4],c[5]+0/1.1]"
    global p225=p[c[0]-0.71*rc,c[1]-0.71*rc,c[2],c[3]+0/1.1,c[4],c[5]+0/1.1]
    $ 383 "p270≔p[c[0],c[1]-rc,c[2],c[3]+0,c[4],c[5]]"
    global p270=p[c[0],c[1]-rc,c[2],c[3]+0,c[4],c[5]]
    $ 384 "p315≔p[c[0]+0.71*rc,c[1]-0.71*rc,c[2],c[3]+0/1.1,c[4],c[5]-0/1.1]"
    global p315=p[c[0]+0.71*rc,c[1]-0.71*rc,c[2],c[3]+0/1.1,c[4],c[5]-0/1.1]
    $ 385 "Set atomization=On"
    set_standard_digital_out(1, True)
    $ 386 "Set triggersolenoid=On"
    set_standard_digital_out(0, True)
    $ 387 "MoveL"
    $ 388 "p0" "breakAfter"
    set_tcp(p[0.0,0.0,0.11,0.0,0.0,0.0])
    movel(p0, a=1.3, v=0.07, r=0.01)
    $ 389 "p45" "breakAfter"
    set_tcp(p[0.0,0.0,0.11,0.0,0.0,0.0])
    movel(p45, a=1.3, v=0.07, r=0.01)
    $ 390 "p90" "breakAfter"
    set_tcp(p[0.0,0.0,0.11,0.0,0.0,0.0])
    movel(p90, a=1.3, v=0.07, r=0.01)
    $ 391 "p135" "breakAfter"
    set_tcp(p[0.0,0.0,0.11,0.0,0.0,0.0])
    movel(p135, a=1.3, v=0.07, r=0.01)
    $ 392 "p180" "breakAfter"
    set_tcp(p[0.0,0.0,0.11,0.0,0.0,0.0])
    movel(p180, a=1.3, v=0.07, r=0.01)
    $ 393 "Set triggersolenoid=Off"
    set_standard_digital_out(0, False)
    $ 394 "Wait: 0.1"
    sleep(0.1)
    $ 395 "Set triggersolenoid=On"
    set_standard_digital_out(0, True)
    $ 396 "p225" "breakAfter"
    set_tcp(p[0.0,0.0,0.11,0.0,0.0,0.0])
    movel(p225, a=1.3, v=0.07, r=0.01)
    $ 397 "p270" "breakAfter"
    set_tcp(p[0.0,0.0,0.11,0.0,0.0,0.0])
    movel(p270, a=1.3, v=0.07, r=0.01)
    $ 398 "p315" "breakAfter"
    set_tcp(p[0.0,0.0,0.11,0.0,0.0,0.0])
    movel(p315, a=1.3, v=0.07, r=0.01)
    $ 399 "p0" "breakAfter"
    set_tcp(p[0.0,0.0,0.11,0.0,0.0,0.0])
    movel(p0, a=1.3, v=0.07, r=0.01)
    $ 400 "p45" "breakAfter"
    set_tcp(p[0.0,0.0,0.11,0.0,0.0,0.0])
    movel(p45, a=1.3, v=0.07, r=0.01)
    $ 401 "Set triggersolenoid=Off"
    set_standard_digital_out(0, False)
    $ 402 "Wait: 0.1"
    sleep(0.1)
    $ 403 "Set triggersolenoid=On"
    set_standard_digital_out(0, True)
    $ 404 "p90" "breakAfter"
    set_tcp(p[0.0,0.0,0.11,0.0,0.0,0.0])
    movel(p90, a=1.3, v=0.07, r=0.01)
    $ 405 "p135" "breakAfter"
    set_tcp(p[0.0,0.0,0.11,0.0,0.0,0.0])
    movel(p135, a=1.3, v=0.07, r=0.01)
    $ 406 "p180" "breakAfter"
    set_tcp(p[0.0,0.0,0.11,0.0,0.0,0.0])
    movel(p180, a=1.3, v=0.07, r=0.01)
    $ 407 "p225" "breakAfter"
    set_tcp(p[0.0,0.0,0.11,0.0,0.0,0.0])
    movel(p225, a=1.3, v=0.07, r=0.01)
    $ 408 "p270" "breakAfter"
    set_tcp(p[0.0,0.0,0.11,0.0,0.0,0.0])
    movel(p270, a=1.3, v=0.07, r=0.01)
    $ 409 "p315" "breakAfter"
    set_tcp(p[0.0,0.0,0.11,0.0,0.0,0.0])
    movel(p315, a=1.3, v=0.07, r=0.01)
    $ 410 "p0" "breakAfter"
    set_tcp(p[0.0,0.0,0.11,0.0,0.0,0.0])
    movel(p0, a=1.3, v=0.07, r=0.01)
    $ 411 "MoveJ"
    $ 412 "Waypoint_15" "breakAfter"
    movej(get_inverse_kin(Waypoint_15_p, qnear=Waypoint_15_q), a=1.3962634015954636, v=1.0471975511965976)
    $ 413 "Wait: 0.2"
    sleep(0.2)
    $ 414 "Set atomization=Off"
    set_standard_digital_out(1, False)
    $ 415 "Set triggersolenoid=Off"
    set_standard_digital_out(0, False)
  end
  def cleaning():
    $ 439 "cleaning" "noBreak"
    $ 440 "MoveJ"
    $ 441 "Waypoint_25" "breakAfter"
    movej(get_inverse_kin(Waypoint_25_p, qnear=Waypoint_25_q), a=1.3962634015954636, v=1.0471975511965976)
    $ 442 "Waypoint_26" "breakAfter"
    movej(get_inverse_kin(Waypoint_26_p, qnear=Waypoint_26_q), a=1.3962634015954636, v=1.0471975511965976)
    $ 443 "Waypoint_27" "breakAfter"
    movej(get_inverse_kin(Waypoint_27_p, qnear=Waypoint_27_q), a=1.3962634015954636, v=1.0471975511965976)
    $ 444 "Waypoint_28" "breakAfter"
    movej(get_inverse_kin(Waypoint_28_p, qnear=Waypoint_28_q), a=1.3962634015954636, v=1.0471975511965976)
    $ 445 "Waypoint_29" "breakAfter"
    movej(get_inverse_kin(Waypoint_29_p, qnear=Waypoint_29_q), a=1.3962634015954636, v=1.0471975511965976)
    $ 446 "Waypoint_30" "breakAfter"
    movej(get_inverse_kin(Waypoint_30_p, qnear=Waypoint_30_q), a=1.3962634015954636, v=1.0471975511965976)
    $ 447 "Waypoint_31" "breakAfter"
    movej(get_inverse_kin(Waypoint_31_p, qnear=Waypoint_31_q), a=1.3962634015954636, v=1.0471975511965976)
    $ 448 "Waypoint_32" "breakAfter"
    movej(get_inverse_kin(Waypoint_32_p, qnear=Waypoint_32_q), a=1.3962634015954636, v=1.0471975511965976)
    $ 449 "Set atomization=On"
    set_standard_digital_out(1, True)
    $ 450 "Set triggersolenoid=On"
    set_standard_digital_out(0, True)
    $ 451 "Wait: 0.2"
    sleep(0.2)
    $ 452 "Set triggersolenoid=Off"
    set_standard_digital_out(0, False)
    $ 453 "Wait: 0.1"
    sleep(0.1)
    $ 454 "Set atomization=Off"
    set_standard_digital_out(1, False)
    $ 455 "Waypoint_33" "breakAfter"
    movej(get_inverse_kin(Waypoint_33_p, qnear=Waypoint_33_q), a=1.3962634015954636, v=1.0471975511965976)
  end
  def turntable():
    $ 456 "turntable" "noBreak"
    $ 457 "MoveJ"
    $ 458 "Waypoint_1" "breakAfter"
    set_tcp(p[0.0,0.0,0.11,0.0,0.0,0.0])
    movej(get_inverse_kin(pose_trans(carouselrod, pose_trans(p[-.225374943892, -.334963115579, .194760490892, -3.139766958285, .106894280104, .000011796367], Waypoint_1_p)), qnear=Waypoint_1_q), a=1.3962634015954636, v=0.5235987755982988, r=0.02)
    $ 459 "Waypoint_2" "breakAfter"
    set_tcp(p[0.0,0.0,0.11,0.0,0.0,0.0])
    movej(get_inverse_kin(pose_trans(carouselrod, pose_trans(p[-.225374943892, -.334963115579, .194760490892, -3.139766958285, .106894280104, .000011796367], Waypoint_2_p)), qnear=Waypoint_2_q), a=1.3962634015954636, v=0.5235987755982988, r=0.02)
    $ 460 "Waypoint_3" "breakAfter"
    set_tcp(p[0.0,0.0,0.11,0.0,0.0,0.0])
    movej(get_inverse_kin(pose_trans(carouselrod, pose_trans(p[-.225374943892, -.334963115579, .194760490892, -3.139766958285, .106894280104, .000011796367], Waypoint_3_p)), qnear=Waypoint_3_q), a=1.3962634015954636, v=0.5235987755982988, r=0.02)
    $ 461 "Waypoint_4" "breakAfter"
    set_tcp(p[0.0,0.0,0.11,0.0,0.0,0.0])
    movej(get_inverse_kin(pose_trans(carouselrod, pose_trans(p[-.225374943892, -.334963115579, .194760490892, -3.139766958285, .106894280104, .000011796367], Waypoint_4_p)), qnear=Waypoint_4_q), a=1.3962634015954636, v=0.5235987755982988, r=0.02)
    $ 462 "Waypoint_5" "breakAfter"
    set_tcp(p[0.0,0.0,0.11,0.0,0.0,0.0])
    movej(get_inverse_kin(pose_trans(carouselrod, pose_trans(p[-.225374943892, -.334963115579, .194760490892, -3.139766958285, .106894280104, .000011796367], Waypoint_5_p)), qnear=Waypoint_5_q), a=1.3962634015954636, v=0.5235987755982988, r=0.02)
    $ 463 "MoveJ"
    $ 464 "Waypoint_6" "breakAfter"
    movej(get_inverse_kin(pose_trans(carouselrod, pose_trans(p[-.225374943892, -.334963115579, .194760490892, -3.139766958285, .106894280104, .000011796367], Waypoint_6_p)), qnear=Waypoint_6_q), a=1.3962634015954636, v=0.3141592653589793)
    $ 465 "Wait: 1.0"
    sleep(1.0)
    $ 466 "MoveJ"
    $ 467 "Waypoint_7" "breakAfter"
    movej(get_inverse_kin(pose_trans(carouselrod, pose_trans(p[-.225374943892, -.334963115579, .194760490892, -3.139766958285, .106894280104, .000011796367], Waypoint_7_p)), qnear=Waypoint_7_q), a=1.3962634015954636, v=1.0471975511965976, r=0.02)
  end
  while (True):
    $ 2 "Robot Program"
    $ 3 "'Program to be used for part #120330-031 rev A BEO beam dump arm'"
    # 'Program to be used for part #120330-031 rev A BEO beam dump arm'
    $ 4 "'Program rev ___: mm/dd/yy note'"
    # 'Program rev ___: mm/dd/yy note'
    $ 5 "timer_1: Start"
    timer_1_is_counting = True
    $ 6 "r≔25/1000"
    global r=25/1000
    $ 7 "A≔30"
    global A=30
    $ 8 "A≔A*3.1416/180"
    global A=A*3.1416/180
    $ 10 "coatnum≔'enter coats'"
    global coatnum=request_integer_from_primary_client("enter coats")
    $ 12 "partnum≔'enter number of parts'"
    global partnum=request_string_from_primary_client("enter number of parts")
    $ 13 "sidenum≔4"
    global sidenum=4
    $ 14 "Loop_1≔1"
    global Loop_1=1
    $ 15 "'NOTE: program not meant to run w/ parts on the side w/ chip and cleaning cup'"
    # 'NOTE: program not meant to run w/ parts on the side w/ chip and cleaning cup'
    $ 131 "If partnum≤sidenum"
    global thread_flag_131=0
    thread Thread_if_131():
      $ 132 "Loop (coatnum)>0"
      thread Thread_while_132():
        while (True):
          $ 133 "partleft≔partnum"
          global partleft=partnum
          $ 134 "loopnum≔1"
          global loopnum=1
          $ 135 "Loop partleft>0"
          thread Thread_while_135():
            while (True):
              $ 136 "If loopnum≟1"
              if (loopnum == 1):
                $ 137 "Call cleaning"
                cleaning()
                $ 138 "Call Spraychip2"
                Spraychip2()
              end
              $ 139 "If loopnum≟1 or loopnum≟5 or loopnum≟9"
              global thread_flag_139=0
              thread Thread_if_139():
                $ 140 "MoveJ"
                $ 141 "c1" "breakAfter"
                movej(get_inverse_kin(c1_p, qnear=c1_q), a=1.3962634015954636, v=1.0471975511965976)
                $ 142 "Set atomization=On"
                set_standard_digital_out(1, True)
                $ 143 "Set triggersolenoid=On"
                set_standard_digital_out(0, True)
                $ 144 "MoveL"
                $ 145 "Waypoint_8" "breakAfter"
                movel(Waypoint_8_p, a=1.2, v=0.2)
                $ 146 "Set triggersolenoid=Off"
                set_standard_digital_out(0, False)
                $ 147 "Wait: 0.1"
                sleep(0.1)
                $ 148 "Set atomization=Off"
                set_standard_digital_out(1, False)
                thread_flag_139 = 1
              end
              if (loopnum == 1  or  loopnum == 5  or  loopnum == 9):
                global thread_handler_139=run Thread_if_139()
                while (thread_flag_139 == 0):
                  if not(loopnum == 1  or  loopnum == 5  or  loopnum == 9):
                    kill thread_handler_139
                    thread_flag_139 = 2
                  else:
                    sync()
                  end
                end
              else:
                thread_flag_139 = 2
              end
              if (thread_flag_139 == 2):
                $ 149 "ElseIf loopnum≟2 or loopnum≟6 or loopnum≟10"
                if (loopnum == 2  or  loopnum == 6  or  loopnum == 10):
                  $ 169 "MoveJ"
                  $ 170 "Waypoint_9" "breakAfter"
                  movej(get_inverse_kin(Waypoint_9_p, qnear=Waypoint_9_q), a=1.3962634015954636, v=1.0471975511965976)
                  $ 171 "Set atomization=On"
                  set_standard_digital_out(1, True)
                  $ 172 "Set triggersolenoid=On"
                  set_standard_digital_out(0, True)
                  $ 173 "MoveL"
                  $ 174 "c2" "breakAfter"
                  movel(c2_p, a=1.2, v=0.2)
                  $ 175 "Set triggersolenoid=Off"
                  set_standard_digital_out(0, False)
                  $ 176 "Wait: 0.1"
                  sleep(0.1)
                  $ 177 "Set atomization=Off"
                  set_standard_digital_out(1, False)
                else:
                  $ 178 "ElseIf loopnum≟3 or loopnum≟7 or loopnum≟11"
                  if (loopnum == 3  or  loopnum == 7  or  loopnum == 11):
                    $ 179 "MoveJ"
                    $ 180 "c3" "breakAfter"
                    movej(get_inverse_kin(c3_p, qnear=c3_q), a=1.3962634015954636, v=1.0471975511965976)
                    $ 181 "Set atomization=On"
                    set_standard_digital_out(1, True)
                    $ 182 "Set triggersolenoid=On"
                    set_standard_digital_out(0, True)
                    $ 183 "MoveL"
                    $ 184 "Waypoint_11" "breakAfter"
                    movel(Waypoint_11_p, a=1.2, v=0.2)
                    $ 185 "Set triggersolenoid=Off"
                    set_standard_digital_out(0, False)
                    $ 186 "Wait: 0.1"
                    sleep(0.1)
                    $ 187 "Set atomization=Off"
                    set_standard_digital_out(1, False)
                  else:
                    $ 188 "Else" "noBreak"
                  end
                end
              end
              $ 209 "loopnum≔loopnum+1"
              global loopnum=loopnum+1
              $ 210 "partleft≔partleft-1"
              global partleft=partleft-1
            end
          end
          if (partleft>0):
            global thread_handler_135=run Thread_while_135()
            while (partleft>0):
              sync()
            end
            kill thread_handler_135
          end
          $ 211 "i≔0"
          global i=0
          $ 212 "coatnum≔coatnum-1"
          global coatnum=coatnum-1
        end
      end
      if ((coatnum)>0):
        global thread_handler_132=run Thread_while_132()
        while ((coatnum)>0):
          sync()
        end
        kill thread_handler_132
      end
      $ 213 "Halt"
      halt
      thread_flag_131 = 1
    end
    if (partnum <= sidenum):
      global thread_handler_131=run Thread_if_131()
      while (thread_flag_131 == 0):
        if not(partnum <= sidenum):
          kill thread_handler_131
          thread_flag_131 = 2
        else:
          sync()
        end
      end
    else:
      thread_flag_131 = 2
    end
    if (thread_flag_131 == 2):
      $ 214 "Else" "noBreak"
      $ 215 "Loop (coatnum)>0"
      thread Thread_while_215():
        while (True):
          $ 216 "partleft≔partnum"
          global partleft=partnum
          $ 217 "loopnum≔1"
          global loopnum=1
          $ 218 "turnnum≔0"
          global turnnum=0
          $ 219 "Loop partleft>0"
          thread Thread_while_219():
            while (True):
              $ 220 "If loopnum≟1"
              if (loopnum == 1):
                $ 221 "Call cleaning"
                cleaning()
                $ 222 "Call Spraychip2"
                Spraychip2()
              end
              $ 223 "If loopnum≟1 or loopnum≟5 or loopnum≟9"
              global thread_flag_223=0
              thread Thread_if_223():
                $ 243 "MoveJ"
                $ 244 "c1" "breakAfter"
                movej(get_inverse_kin(c1_p, qnear=c1_q), a=1.3962634015954636, v=1.0471975511965976)
                $ 245 "Set atomization=On"
                set_standard_digital_out(1, True)
                $ 246 "Set triggersolenoid=On"
                set_standard_digital_out(0, True)
                $ 247 "MoveL"
                $ 248 "Waypoint_8" "breakAfter"
                movel(Waypoint_8_p, a=1.2, v=0.2)
                $ 249 "Set triggersolenoid=Off"
                set_standard_digital_out(0, False)
                $ 250 "Wait: 0.1"
                sleep(0.1)
                $ 251 "Set atomization=Off"
                set_standard_digital_out(1, False)
                thread_flag_223 = 1
              end
              if (loopnum == 1  or  loopnum == 5  or  loopnum == 9):
                global thread_handler_223=run Thread_if_223()
                while (thread_flag_223 == 0):
                  if not(loopnum == 1  or  loopnum == 5  or  loopnum == 9):
                    kill thread_handler_223
                    thread_flag_223 = 2
                  else:
                    sync()
                  end
                end
              else:
                thread_flag_223 = 2
              end
              if (thread_flag_223 == 2):
                $ 252 "ElseIf loopnum≟2 or loopnum≟6 or loopnum≟10"
                if (loopnum == 2  or  loopnum == 6  or  loopnum == 10):
                  $ 272 "MoveJ"
                  $ 273 "Waypoint_9" "breakAfter"
                  movej(get_inverse_kin(Waypoint_9_p, qnear=Waypoint_9_q), a=1.3962634015954636, v=1.0471975511965976)
                  $ 274 "Set atomization=On"
                  set_standard_digital_out(1, True)
                  $ 275 "Set triggersolenoid=On"
                  set_standard_digital_out(0, True)
                  $ 276 "MoveL"
                  $ 277 "c2" "breakAfter"
                  movel(c2_p, a=1.2, v=0.2)
                  $ 278 "Set triggersolenoid=Off"
                  set_standard_digital_out(0, False)
                  $ 279 "Wait: 0.1"
                  sleep(0.1)
                  $ 280 "Set atomization=Off"
                  set_standard_digital_out(1, False)
                else:
                  $ 281 "ElseIf loopnum≟3 or loopnum≟7 or loopnum≟11"
                  if (loopnum == 3  or  loopnum == 7  or  loopnum == 11):
                    $ 282 "MoveJ"
                    $ 283 "c3" "breakAfter"
                    movej(get_inverse_kin(c3_p, qnear=c3_q), a=1.3962634015954636, v=1.0471975511965976)
                    $ 284 "Set atomization=On"
                    set_standard_digital_out(1, True)
                    $ 285 "Set triggersolenoid=On"
                    set_standard_digital_out(0, True)
                    $ 286 "MoveL"
                    $ 287 "Waypoint_11" "breakAfter"
                    movel(Waypoint_11_p, a=1.2, v=0.2)
                    $ 288 "Set triggersolenoid=Off"
                    set_standard_digital_out(0, False)
                    $ 289 "Wait: 0.1"
                    sleep(0.1)
                    $ 290 "Set atomization=Off"
                    set_standard_digital_out(1, False)
                  else:
                    $ 291 "Else" "noBreak"
                    $ 312 "MoveJ"
                    $ 313 "Waypoint_10" "breakAfter"
                    movej(get_inverse_kin(Waypoint_10_p, qnear=Waypoint_10_q), a=1.3962634015954636, v=1.0471975511965976)
                    $ 314 "Set atomization=On"
                    set_standard_digital_out(1, True)
                    $ 315 "Set triggersolenoid=On"
                    set_standard_digital_out(0, True)
                    $ 316 "MoveL"
                    $ 317 "c4" "breakAfter"
                    movel(c4_p, a=1.2, v=0.2)
                    $ 318 "Set triggersolenoid=Off"
                    set_standard_digital_out(0, False)
                    $ 319 "Wait: 0.1"
                    sleep(0.1)
                    $ 320 "Set atomization=Off"
                    set_standard_digital_out(1, False)
                  end
                end
              end
              $ 321 "loopnum≔loopnum+1"
              global loopnum=loopnum+1
              $ 322 "partleft≔partleft-1"
              global partleft=partleft-1
            end
          end
          if (partleft>0):
            global thread_handler_219=run Thread_while_219()
            while (partleft>0):
              sync()
            end
            kill thread_handler_219
          end
          $ 323 "i≔0"
          global i=0
          $ 324 "Loop (6-turnnum)>0"
          thread Thread_while_324():
            while (True):
              $ 325 "Call turntable"
              turntable()
              $ 326 "turnnum≔turnnum+1"
              global turnnum=turnnum+1
            end
          end
          if ((6-turnnum)>0):
            global thread_handler_324=run Thread_while_324()
            while ((6-turnnum)>0):
              sync()
            end
            kill thread_handler_324
          end
          $ 327 "coatnum≔coatnum-1"
          global coatnum=coatnum-1
        end
      end
      if ((coatnum)>0):
        global thread_handler_215=run Thread_while_215()
        while ((coatnum)>0):
          sync()
        end
        kill thread_handler_215
      end
      $ 328 "Halt"
      halt
    end
  end
end
